PROGRAM MAIN
VAR
	fbMath	:FB_Math;
	icnt	:UDINT;
END_VAR

icnt:=icnt+1;

END_PROGRAM

(* stored: Version 1.1.0.1, ProductVersion 3.1.4024.9
   POU MAIN: Id {5af3ba7a-78d9-4457-8427-585f93cb09e4}, SpecialFunc None *)
